{attribute 'qualified_only'}
VAR_GLOBAL
	iInput1 AT %I* : INT;
END_VAR

(* stored: Version 1.1.0.1, ProductVersion 3.1.4024.11
   GVL MyGVL: Id {f330120a-278f-47ab-823f-0ceb72bcac09} *)
